(* CODESYS project SM_IND.library
   Description: Device support for Industrial Automation board under Raspberry Pi
   Version: 1.1.0.0
   Title: Raspberry I2C INDUSTRIAL AUTOMATION
   Company: Sequent Microsystems
   DocFormat: reStructuredText
   Placeholder: PlaceholderTemplate
   LanguageModelAttribute: qualified-access-only
   Author: Sequent Microsystems
   DefaultNamespace: SM_IND

Project tree, tasks and I/O mapping:
  libraries: Raspberry Pi Peripherals, 4.6.0.0 (3S - Smart Software Solutions GmbH); IoStandard, 3.5.17.0 (System); Standard, 3.5.18.0 (System)
  global variables GVL
  function block SM_IND [ST]: AfterReadInputs, BeforeWriteOutputs
  Library Information/
    function GetLibVersionNumber [ST]
    function GetLibVersion [ST]
    function IsLibReleased [ST]
  Project Information/
    function GetCompany [ST]
    function GetTitle [ST]
    function GetVersion [ST]
    function GetTextProperty [ST]
    function GetTextProperty2 [ST]
    function GetNumberProperty [ST]
    function GetBooleanProperty [ST]
    function GetVersionProperty [ST]
*)

// GVL
//{attribute 'qualified_only'}
VAR_GLOBAL CONSTANT
	LED_VAL_ADD: USINT := 16#00;
	LED_SET_ADD: USINT := 16#01;
	LED_CLR_ADD: USINT := 16#02;
	OPTO_VAL_ADD: USINT := 16#03;
	
	I4_20_OUT_VAL1_ADD: USINT := 16#0C;
	I4_20_IN_VAL1_ADD: USINT := 16#2C;
	U0_10_OUT_VAL1_ADD: USINT := 16#04;
	U0_10_IN_VAL1_ADD: USINT := 16#1C;
	OD_PWM1_ADD:USINT:= 16#14;
	TEMPERATURE_ADD: USINT := 16#27;
	OWB_DEV_COUNT_ADD: USINT := 16#93;
	OWB_TEMP1_ADD: USINT := 16#AE;
	
END_VAR

// SM_IND
FUNCTION_BLOCK SM_IND EXTENDS i2c
VAR_INPUT
	ledState: ARRAY[0..3] OF BOOL;
	out0_10Volt: ARRAY[0..3] OF REAL;
	out4_20Ma: ARRAY[0..3] OF REAL;
	outOdPwm:ARRAY[0..3] OF REAL;
END_VAR
VAR_OUTPUT
	inOpto: ARRAY[0..3] OF BOOL;
	in0_10Volt: ARRAY[0..3] OF REAL;
	in4_20Ma: ARRAY[0..3] OF REAL;
	inOWBTemp: ARRAY[0..15] OF REAL;
	inOWBSensors: USINT;
	boardTemperature: REAL;
END_VAR
VAR
	timer: TON := (IN:=TRUE);
	ledStateRaw: USINT;
	out0_10VoltRaw: ARRAY[0..3] OF UINT;
	out4_20MaRaw: ARRAY[0..3] OF UINT;
	outOdPwmRaw: ARRAY[0..3] OF UINT;
	readOWBCount: USINT;
END_VAR
VAR_TEMP	
	i, usi: USINT;
	buff: ARRAY[0..20] OF USINT;	
END_VAR

SUPER^();

CASE _iState OF
0:
	IF usiAddress < 16#50 OR  usiAddress > 16#58 THEN
		usiAddress := 16#50;
	END_IF
	//usiAddress := 16#31 + StackLevel;
	IF SUPER^.init() THEN
		_iState := 5;
	END_IF	
5:	
	Timer.pt := T#20MS;
	buff[1] := 0;
	buff[2] := 0;
	FOR i:=0 TO 3 DO
		buff[0] := I4_20_OUT_VAL1_ADD + i* 2;	
  		write(ADR(buff), 3);
		out4_20MaRaw[i] := 0;
		
		buff[0] := U0_10_OUT_VAL1_ADD + i* 2;
		write(ADR(buff), 3);
		out0_10VoltRaw[i] := 0;
	END_FOR
	
	// init all relay off
	
	ledStateRaw := 0;
	write8(LED_VAL_ADD, 0);
	readOWBCount:=0;
	
	_iState := 10;
END_CASE

METHOD AfterReadInputs:INT
VAR
	Buffer : ARRAY[0..3] OF BYTE;
	ch: USINT;
	address: USINT;
	value: REAL;
	len: DINT;	
	opto: USINT;
END_VAR
SUPER^.AfterReadInputs();

IF _iState = 10 THEN
	timer(IN:=TRUE);
	IF timer.Q THEN	
		opto := read8(OPTO_VAL_ADD);  
		FOR len:=0 TO 3 DO
			inOpto[len] := USINT_TO_BOOL(SHL(2#00000001, len) AND opto);
		END_FOR
	
		boardTemperature := read8(TEMPERATURE_ADD)/10;
		IF readOWBCount < 50 THEN
			readOWBCount := readOWBCount + 1;	
		ELSE
			readOWBCount := 0;
			inOWBSensors := read8(OWB_DEV_COUNT_ADD);	
			IF inOWBSensors > 0 THEN
				FOR ch:=0 TO inOWBSensors - 1 DO
					address:= OWB_TEMP1_ADD + 2*ch;
					len := readregister(address, ADR(Buffer), 2);		
					IF len = 2 THEN
						value := BYTE_TO_REAL(Buffer[0]) + BYTE_TO_REAL(Buffer[1]) * 256;
						inOWBTemp[ch]:=value/100;
					END_IF
				END_FOR
			END_IF
		END_IF
	
		FOR ch:=0 TO 3 DO
			address:= I4_20_IN_VAL1_ADD + 2*ch;
			len := readregister(address, ADR(Buffer), 2);		
			IF len = 2 THEN
				value := BYTE_TO_REAL(Buffer[0]) + BYTE_TO_REAL(Buffer[1]) * 256;
				in4_20Ma[ch]:=value/1000;
			END_IF
		END_FOR
		FOR ch:=0 TO 3 DO
			address:= U0_10_IN_VAL1_ADD + 2*ch;
			len := readregister(address, ADR(Buffer), 2);		
			IF len = 2 THEN
				value := BYTE_TO_REAL(Buffer[0]) + BYTE_TO_REAL(Buffer[1]) * 256;
				in0_10Volt[ch]:=value/1000;
			END_IF
		END_FOR
		
		timer(IN:=FALSE);
	END_IF
END_IF
END_METHOD

METHOD BeforeWriteOutputs:INT
VAR
	i: USINT;
	cnt: USINT;
	inVal:UINT;
	inSVal:USINT;
	buff: ARRAY[0..2] OF USINT;
	wStat: BOOL;
END_VAR
SUPER^.BeforeWriteOutputs();

IF _iState = 10 THEN
	
	FOR i:=0 TO 3 DO
		IF out4_20Ma[i] < 4 THEN
			out4_20Ma[i] := 4;
		END_IF
		IF out4_20Ma[i] > 20 THEN
			out4_20Ma[i] := 20;
		END_IF
		inVal := REAL_TO_UINT(out4_20Ma[i] * 1000);
		IF out4_20MaRaw[i] <> inVal THEN
			buff[0] := I4_20_OUT_VAL1_ADD + 2*i;
			buff[2] := UINT_TO_USINT(inVal / 256);
			buff[1] := UINT_TO_USINT(inVal - (inVal / 256));
			cnt := DINT_TO_USINT(write(ADR(buff), 3));
			IF cnt = 3 THEN
				out4_20MaRaw[i] := inVal;
			END_IF	
		END_IF
	END_FOR
	
	FOR i:=0 TO 3 DO
		IF out0_10Volt[i] < 0 THEN
			out0_10Volt[i] := 0;
		END_IF
		IF out0_10Volt[i] > 10 THEN
			out0_10Volt[i] := 10;
		END_IF
		inVal := REAL_TO_UINT(out0_10Volt[i] * 1000);
		IF out0_10VoltRaw[i] <> inVal THEN
			buff[0] := U0_10_OUT_VAL1_ADD + 2*i;
			buff[2] := UINT_TO_USINT(inVal / 256);
			buff[1] := UINT_TO_USINT(inVal - (inVal / 256));
			cnt := DINT_TO_USINT(write(ADR(buff), 3));
			IF cnt = 3 THEN
				out0_10VoltRaw[i] := inVal;
			END_IF	
		END_IF
	END_FOR  
	
	FOR i:=0 TO 3 DO
		IF outOdPwm[i] < 0 THEN
			outOdPwm[i] := 0;
		END_IF
		IF outOdPwm[i] > 100 THEN
			outOdPwm[i] := 100;
		END_IF
		inVal := REAL_TO_UINT(outOdPwm[i] * 100);
		IF outOdPwmRaw[i] <> inVal THEN
			buff[0] := OD_PWM1_ADD + 2*i;
			buff[2] := UINT_TO_USINT(inVal / 256);
			buff[1] := UINT_TO_USINT(inVal - (inVal / 256));
			cnt := DINT_TO_USINT(write(ADR(buff), 3));
			IF cnt = 3 THEN
				outOdPwmRaw[i] := inVal;
			END_IF	
		END_IF
	END_FOR  
	
	inSVal:= 0;
	FOR i:= 0 TO 3 DO
		inSVal:= inSVal + SHL(BOOL_TO_USINT(ledState[i]), i +4);
	END_FOR
	IF ledStateRaw <> inSVal THEN
		IF write8(LED_VAL_ADD, inSVal) THEN
			ledStateRaw:=inSVal;
		END_IF
	END_IF		
END_IF
END_METHOD

END_FUNCTION_BLOCK

// Library Information/GetLibVersionNumber
// This function has been automatically generated from the project information.
FUNCTION GetLibVersionNumber : DWORD
VAR_INPUT
	
END_VAR

GetLibVersionNumber := 16842752;

END_FUNCTION

// Project Information/GetCompany
// This function has been automatically generated from the project information.
{attribute 'signature_flag' := '1073741824'}
{attribute 'register_in_runtime'}
FUNCTION GetCompany : WSTRING
VAR_INPUT
	
END_VAR

GetCompany := "Sequent Microsystems";

END_FUNCTION

// Project Information/GetTitle
// This function has been automatically generated from the project information.
{attribute 'signature_flag' := '1073741824'}
{attribute 'register_in_runtime'}
FUNCTION GetTitle : WSTRING
VAR_INPUT
	
END_VAR

GetTitle := "Raspberry I2C INDUSTRIAL AUTOMATION";

END_FUNCTION

// Library Information/GetLibVersion
// This function has been automatically generated from the project information.
FUNCTION GetLibVersion : VERSION
VAR_INPUT
	
END_VAR

GetLibVersion.uiMajor := 1;
GetLibVersion.uiMinor := 1;
GetLibVersion.uiServicePack := 0;
GetLibVersion.uiPatch := 0;

END_FUNCTION

// Library Information/IsLibReleased
// This function has been automatically generated from the project information.
FUNCTION IsLibReleased : BOOL
VAR_INPUT
	
END_VAR

IsLibReleased := FALSE;

END_FUNCTION

// Project Information/GetVersion
// This function has been automatically generated from the project information.
{attribute 'signature_flag' := '1073741824'}
{attribute 'register_in_runtime'}
FUNCTION GetVersion : VERSION
VAR_INPUT
	
END_VAR

GetVersion.uiMajor := 1;
GetVersion.uiMinor := 1;
GetVersion.uiServicePack := 0;
GetVersion.uiPatch := 0;

END_FUNCTION

// Project Information/GetTextProperty
// This function has been automatically generated from the project information.
{attribute 'signature_flag' := '1073741824'}
{attribute 'register_in_runtime'}
FUNCTION GetTextProperty : WSTRING
VAR_INPUT
	stKey: WSTRING;
END_VAR

IF stKey = "Author" THEN
	GetTextProperty := "Sequent Microsystems";
ELSIF stKey = "Company" THEN
	GetTextProperty := "Sequent Microsystems";
ELSIF stKey = "DefaultNamespace" THEN
	GetTextProperty := "SM_IND";
ELSIF stKey = "Description" THEN
	GetTextProperty := "Device support for Industrial Automation board under Raspberry Pi";
ELSIF stKey = "DocFormat" THEN
	GetTextProperty := "reStructuredText";
ELSIF stKey = "LanguageModelAttribute" THEN
	GetTextProperty := "qualified-access-only";
ELSIF stKey = "Placeholder" THEN
	GetTextProperty := "PlaceholderTemplate";
ELSIF stKey = "Project" THEN
	GetTextProperty := "SM_IND";
ELSIF stKey = "Title" THEN
	GetTextProperty := "Raspberry I2C INDUSTRIAL AUTOMATION";
ELSE
	GetTextProperty := "";
END_IF

END_FUNCTION

// Project Information/GetTextProperty2
// This function has been automatically generated from the project information.
{attribute 'signature_flag' := '1073741824'}
{attribute 'register_in_runtime'}
FUNCTION GetTextProperty2 : POINTER TO WSTRING
VAR_INPUT
	stKey: WSTRING;
END_VAR

IF stKey = "Author" THEN
	GetTextProperty2 := ADR("Sequent Microsystems");
ELSIF stKey = "Company" THEN
	GetTextProperty2 := ADR("Sequent Microsystems");
ELSIF stKey = "DefaultNamespace" THEN
	GetTextProperty2 := ADR("SM_IND");
ELSIF stKey = "Description" THEN
	GetTextProperty2 := ADR("Device support for Industrial Automation board under Raspberry Pi");
ELSIF stKey = "DocFormat" THEN
	GetTextProperty2 := ADR("reStructuredText");
ELSIF stKey = "LanguageModelAttribute" THEN
	GetTextProperty2 := ADR("qualified-access-only");
ELSIF stKey = "Placeholder" THEN
	GetTextProperty2 := ADR("PlaceholderTemplate");
ELSIF stKey = "Project" THEN
	GetTextProperty2 := ADR("SM_IND");
ELSIF stKey = "Title" THEN
	GetTextProperty2 := ADR("Raspberry I2C INDUSTRIAL AUTOMATION");
ELSE
	GetTextProperty2 := ADR("");
END_IF

END_FUNCTION

// Project Information/GetNumberProperty
// This function has been automatically generated from the project information.
{attribute 'signature_flag' := '1073741824'}
{attribute 'register_in_runtime'}
FUNCTION GetNumberProperty : DINT
VAR_INPUT
	stKey: WSTRING;
END_VAR

GetNumberProperty := 0;

END_FUNCTION

// Project Information/GetBooleanProperty
// This function has been automatically generated from the project information.
{attribute 'signature_flag' := '1073741824'}
{attribute 'register_in_runtime'}
FUNCTION GetBooleanProperty : BOOL
VAR_INPUT
	stKey: WSTRING;
END_VAR

IF stKey = "IsEndUserLibrary" THEN
	GetBooleanProperty := FALSE;
ELSIF stKey = "Released" THEN
	GetBooleanProperty := FALSE;
ELSE
	GetBooleanProperty := FALSE;
END_IF

END_FUNCTION

// Project Information/GetVersionProperty
// This function has been automatically generated from the project information.
{attribute 'signature_flag' := '1073741824'}
{attribute 'register_in_runtime'}
FUNCTION GetVersionProperty : VERSION
VAR_INPUT
	stKey: WSTRING;
END_VAR

IF stKey = "Version" THEN
	GetVersionProperty.uiMajor := 1;
	GetVersionProperty.uiMinor := 1;
	GetVersionProperty.uiServicePack := 0;
	GetVersionProperty.uiPatch := 0;
ELSE
	GetVersionProperty.uiMajor := 0;
	GetVersionProperty.uiMinor := 0;
	GetVersionProperty.uiServicePack := 0;
	GetVersionProperty.uiPatch := 0;
END_IF

END_FUNCTION
